// SIMATIC STEP 7 (V5.x) project Gradirn
// CPU: CPU 315-2PN/DP
// station: Hardware
// station: SIMATIC 300(1)
// station: P_ADR_BUS
// station: P_ADR_BUS
// station: Configuration
// program: S7 Program(3)

SYMBOL_TABLE
""		
"grad_motor_1"	DB 1	FB 41
"grad_motor_2"	DB 2	FB 41
"Alarms"	DB 3	DB 3
"values"	DB 4	DB 4
"Data_motors"	DB 5	FB 4
"Motor_grad"	FB 1	FB 1	// Вентилятор градирни
"Motors"	FB 4	FB 4
"CONT_C"	FB 41	FB 41	// Continuous Control
"CONT_S"	FB 42	FB 42	// Step Control
"TCONT_CP"	FB 58	FB 58	// temperature PID controller with pulse generator and self-tuning
"TCONT_S"	FB 59	FB 59	// temperature PID step controller
"Level_grad"	FC 1	FC 1
"read/write values"	FC 2	FC 2
"Fault_motor"	FC 3	FC 3
"Pumps"	FC 4	FC 4
"Alarm"	FC 5	FC 5
"S5TI_TIM"	FC 33	FC 33	// S5 Time to IEC Time
"TIM_S5TI"	FC 40	FC 40	// IEC Time to S5 Time
"Read Analog Value 464-1"	FC 104	FC 104	// Read Analog Value 464-1
"Read Analog Value 464-2"	FC 105	FC 105	// Read Analog Value 464-2
"mode_man_V1"	M 0.0	BOOL
"valve_out"	M 2.0	BOOL
"valve_opened"	M 2.1	BOOL
"valve_closed"	M 2.2	BOOL
"always_on"	M 6.0	BOOL	// всегда 1
"V1_btn_pusk"	M 100.0	BOOL
"V1_btn_stop"	M 100.1	BOOL
"V1_inverter_ok"	M 100.2	BOOL
"V1_mode_remote"	M 100.3	BOOL
"V1_start"	M 100.4	BOOL
"V1_error"	M 100.5	BOOL
"V1_loc_p"	M 100.6	BOOL
"V1_loc_st"	M 100.7	BOOL
"V2_btn_pusk"	M 101.0	BOOL
"V2_btn_stop"	M 101.1	BOOL
"V2_inverter_ok"	M 101.2	BOOL
"V2_mode_remote"	M 101.3	BOOL
"V2_start"	M 101.4	BOOL
"V2_error"	M 101.5	BOOL
"V2_loc_p"	M 101.6	BOOL
"V2_loc_st"	M 101.7	BOOL
"on_H1"	M 102.0	BOOL
"on_H2"	M 102.1	BOOL
"psal_H1"	M 102.2	BOOL
"psal_H2"	M 102.3	BOOL
"tsah_H1"	M 102.4	BOOL
"tsah_H2"	M 102.5	BOOL
"H1_PU"	M 102.6	BOOL
"H1_ST"	M 102.7	BOOL
"H1_MD"	M 103.0	BOOL
"H2_PU"	M 103.1	BOOL
"H2_ST"	M 103.2	BOOL
"H2_MD"	M 103.3	BOOL
"rez_H1"	M 103.4	BOOL
"rez_H2"	M 103.5	BOOL
"btn_H1_PU"	M 103.6	BOOL
"btn_H1_ST"	M 103.7	BOOL
"btn_H2_PU"	M 104.0	BOOL
"btn_H2_ST"	M 104.1	BOOL
"V1_running"	M 110.0	BOOL
"V2_running"	M 111.1	BOOL
"V1_Gain"	MD 2	REAL
"V1_I"	MD 6	TIME
"V1_SP"	MD 10	REAL
"V1_out_freq"	MD 14	REAL
"Temp_grad"	MD 18	REAL
"V1_MAN_SP"	MD 22	REAL
"V_cycle"	MD 26	TIME
"main"	OB 1	OB 1
"pid"	OB 35	OB 35
"TON"	SFB 4	SFB 4	// Generate an On Delay
"Analog values insert"	UDT 1	UDT 1
END_SYMBOL_TABLE

FUNCTION_BLOCK "Motor_grad"	// FB 1
VERSION : 0.1
VAR_INPUT
  btn_pusk : BOOL ;
  btn_stop : BOOL ;
  mode_remote : BOOL ;
  inverter_ok : BOOL ;
  motor_error : BOOL ;
  loc_pusk : BOOL ;
  loc_stop : BOOL ;
  tim_1 : TIMER ;
  tim_2 : TIMER ;
END_VAR
VAR_OUTPUT
  motor_start : BOOL ;
END_VAR
BEGIN
NETWORK
TITLE = start
      A     #inverter_ok;
      A     #mode_remote;
      A     #btn_pusk;
      O(;
      AN    #mode_remote;
      A     #inverter_ok;
      A     #loc_pusk;
      L     S5T#400MS;
      T     LD 0;
      TAK;
      T     LD 4;
      L     #tim_1;
      T     LW 8;
      L     LD 4;
      L     LD 0;
      SD    T [LW 8];
      T     LD 0;
      TAK;
      T     LD 4;
      L     #tim_1;
      T     LW 8;
      L     LD 4;
      L     LD 0;
      A     T [LW 8];
      );
      S     #motor_start;
NETWORK
TITLE = stop
      ON    #inverter_ok;
      O     #motor_error;
      O(;
      A     #mode_remote;
      A     #btn_stop;
      );
      O(;
      L     S5T#400MS;
      AN    #mode_remote;
      A     #loc_stop;
      T     LD 0;
      TAK;
      T     LD 4;
      L     #tim_2;
      T     LW 8;
      L     LD 4;
      L     LD 0;
      SD    T [LW 8];
      T     LD 0;
      TAK;
      T     LD 4;
      L     #tim_2;
      T     LW 8;
      L     LD 4;
      L     LD 0;
      A     T [LW 8];
      );
      R     #motor_start;
END_FUNCTION_BLOCK

FUNCTION_BLOCK "Motors"	// FB 4
VERSION : 0.1
VAR
  mifb_1 : FB 1;
  mifb_2 : FB 1;
END_VAR
BEGIN
NETWORK
TITLE =
      CALL  #mifb_1 (
           btn_pusk                 := "V1_btn_pusk",
           btn_stop                 := "V1_btn_stop",
           mode_remote              := "V1_mode_remote",
           inverter_ok              := "V1_inverter_ok",
           motor_error              := "V1_error",
           loc_pusk                 := "V1_loc_p",
           loc_stop                 := "V1_loc_st",
           tim_1                    := T 1,
           tim_2                    := T 2,
           motor_start              := "V1_start");
NETWORK
TITLE =
      CALL  #mifb_2 (
           btn_pusk                 := "V2_btn_pusk",
           btn_stop                 := "V2_btn_stop",
           mode_remote              := "V2_mode_remote",
           inverter_ok              := "V2_inverter_ok",
           motor_error              := "V2_error",
           loc_pusk                 := "V2_loc_p",
           loc_stop                 := "V2_loc_st",
           tim_1                    := T 3,
           tim_2                    := T 4,
           motor_start              := "V2_start");
END_FUNCTION_BLOCK

// FB 41: know-how protected block, not included

FUNCTION "Level_grad" : VOID	// FC 1
TITLE = Fulling level grad
VERSION : 0.1
BEGIN
NETWORK
TITLE =
      L     "values".level_grad;
      L     "values".level_sp;
      <R;
      JC    open;
      R     "valve_out";
      JU    end;
open: S     "valve_out";
end:  NOP   0;
END_FUNCTION

FUNCTION "read/write values" : VOID	// FC 2
VERSION : 0.1
BEGIN
NETWORK
TITLE =
      A     "values".zero;
      =     L 0.0;
      BLD   103;
      CALL  "Read Analog Value 464-2" (
           $1                       := P#P 256.0,
           $2                       := "values".hi_temp_grad,
           $3                       := "values".low_temp_grad,
           $4                       := L 0.0,
           $5                       := "values".error_temp_grad,
           $6                       := "values".temp_grad);
      NOP   0;
NETWORK
TITLE =
      A     "values".zero;
      =     L 0.0;
      BLD   103;
      CALL  "Read Analog Value 464-2" (
           $1                       := P#P 272.0,
           $2                       := "values".level_hi,
           $3                       := "values".level_low,
           $4                       := L 0.0,
           $5                       := "values".error_level,
           $6                       := "values".level_grad);
      NOP   0;
NETWORK
TITLE = read vibrations motors
      A     "values".zero;
      =     L 0.0;
      BLD   103;
      CALL  "Read Analog Value 464-2" (
           $1                       := P#P 274.0,
           $2                       := "values".vibr_1_hi,
           $3                       := "values".vibr_1_low,
           $4                       := L 0.0,
           $5                       := "values".vibr_1_er,
           $6                       := "values".vibr_1);
      NOP   0;
NETWORK
TITLE =
      A     "values".zero;
      =     L 0.0;
      BLD   103;
      CALL  "Read Analog Value 464-2" (
           $1                       := P#P 276.0,
           $2                       := "values".vibr_1_hi,
           $3                       := "values".vibr_1_low,
           $4                       := L 0.0,
           $5                       := "values".vibr_2_er,
           $6                       := "values".vibr_2);
      NOP   0;
NETWORK
TITLE = Current V1
      CALL  "Read Analog Value 464-2" (
           $1                       := P#P 278.0,
           $2                       := "values".curr_1_hi,
           $3                       := "values".curr_1_low,
           $4                       := "values".zero,
           $5                       := "values".curr_1_er,
           $6                       := "values".curr_1);
NETWORK
TITLE = Current V2
      CALL  "Read Analog Value 464-2" (
           $1                       := P#P 280.0,
           $2                       := "values".curr_1_hi,
           $3                       := "values".curr_1_low,
           $4                       := "values".zero,
           $5                       := "values".curr_2_er,
           $6                       := "values".curr_2);
NETWORK
TITLE = discret inputs/outputs V1,V2
      A     I 8.0;
      =     "V1_loc_p";
      A     I 8.1;
      =     "V1_loc_st";
      A     I 8.2;
      =     "V1_inverter_ok";
      A     "V1_start";
      =     Q 11.0;
      A     I 8.3;
      =     "V1_mode_remote";
      A     I 8.4;
      =     "V1_running";
      A     I 9.0;
      =     "V2_loc_p";
      A     I 9.1;
      =     "V2_loc_st";
      A     I 9.2;
      =     "V2_inverter_ok";
      A     "V2_start";
      =     Q 11.1;
      A     I 9.3;
      =     "V2_mode_remote";
      A     I 9.4;
      =     "V2_running";
NETWORK
TITLE = Pump signals
      A     I 10.0;
      =     "on_H1";
      A     I 10.1;
      =     "on_H2";
      A     I 10.2;
      =     "psal_H1";
      A     I 10.3;
      =     "psal_H2";
      A     I 10.4;
      =     "tsah_H1";
      A     I 10.5;
      =     "tsah_H2";
      A     "H1_PU";
      =     Q 11.2;
      A     "H1_ST";
      =     Q 11.3;
      A     "H1_MD";
      =     Q 11.4;
      A     "H2_PU";
      =     Q 11.5;
      A     "H2_ST";
      =     Q 11.6;
      A     "H2_MD";
      =     Q 11.7;
NETWORK
TITLE =
      CALL  "Read Analog Value 464-2" (
           $1                       := P#P 282.0,
           $2                       := "values".curr_1_hi,
           $3                       := "values".curr_1_low,
           $4                       := "values".zero,
           $5                       := "values".curr_H1_er,
           $6                       := "values".curr_H1);
      CALL  "Read Analog Value 464-2" (
           $1                       := P#P 284.0,
           $2                       := "values".curr_1_hi,
           $3                       := "values".curr_1_low,
           $4                       := "values".zero,
           $5                       := "values".curr_H2_er,
           $6                       := "values".curr_2);
END_FUNCTION

FUNCTION "Fault_motor" : VOID	// FC 3
VERSION : 0.1
BEGIN
NETWORK
TITLE = fault motor 1 of vibration
      L     "values".vibr_1;
      L     1.200000e+01;
      >R;
      =     "V1_error";
NETWORK
TITLE =
      L     "values".vibr_2;
      L     1.200000e+01;
      >R;
      =     "V2_error";
END_FUNCTION

FUNCTION "Pumps" : VOID	// FC 4
VERSION : 0.1
VAR_TEMP
  fl_1 : BOOL ;
  fl_2 : BOOL ;
  tr_1 : BOOL ;
END_VAR
BEGIN
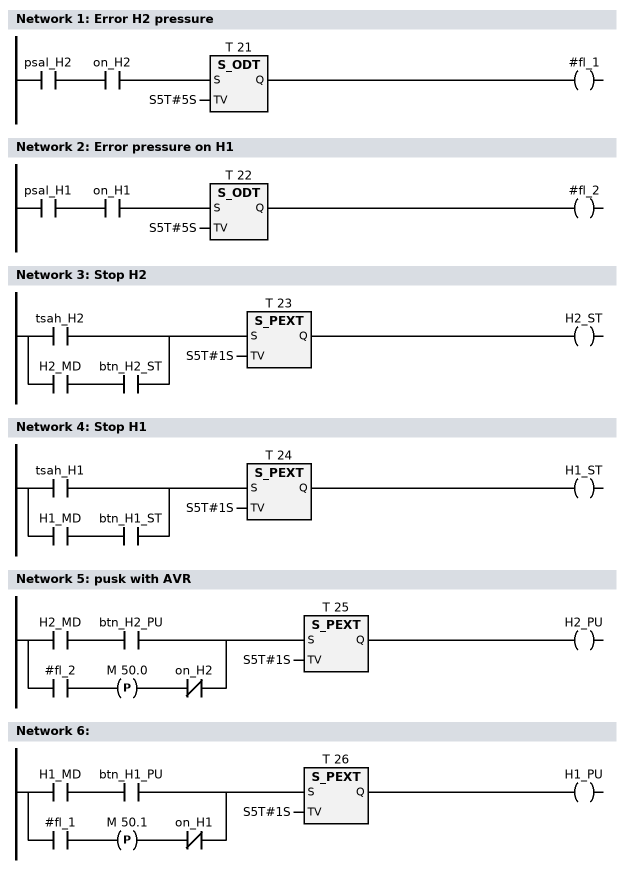
NETWORK
TITLE = Error H2 pressure
      A     "psal_H2";
      A     "on_H2";
      L     S5T#5S;
      SD    T 21;
      NOP   0;
      NOP   0;
      NOP   0;
      A     T 21;
      =     #fl_1;
NETWORK
TITLE = Error pressure on H1
      A     "psal_H1";
      A     "on_H1";
      L     S5T#5S;
      SD    T 22;
      NOP   0;
      NOP   0;
      NOP   0;
      A     T 22;
      =     #fl_2;
NETWORK
TITLE = Stop H2
      A(;
      O     "tsah_H2";
      O;
      A     "H2_MD";
      A     "btn_H2_ST";
      );
      L     S5T#1S;
      SE    T 23;
      NOP   0;
      NOP   0;
      NOP   0;
      A     T 23;
      =     "H2_ST";
NETWORK
TITLE = Stop H1
      A(;
      O     "tsah_H1";
      O;
      A     "H1_MD";
      A     "btn_H1_ST";
      );
      L     S5T#1S;
      SE    T 24;
      NOP   0;
      NOP   0;
      NOP   0;
      A     T 24;
      =     "H1_ST";
NETWORK
TITLE = pusk with AVR
      A(;
      A     "H2_MD";
      A     "btn_H2_PU";
      O(;
      A     #fl_2;
      FP    M 50.0;
      AN    "on_H2";
      );
      );
      L     S5T#1S;
      SE    T 25;
      NOP   0;
      NOP   0;
      NOP   0;
      A     T 25;
      =     "H2_PU";
NETWORK
TITLE =
      A(;
      A     "H1_MD";
      A     "btn_H1_PU";
      O(;
      A     #fl_1;
      FP    M 50.1;
      AN    "on_H1";
      );
      );
      L     S5T#1S;
      SE    T 26;
      NOP   0;
      NOP   0;
      NOP   0;
      A     T 26;
      =     "H1_PU";
END_FUNCTION

FUNCTION "Alarm" : VOID	// FC 5
VERSION : 0.1
BEGIN
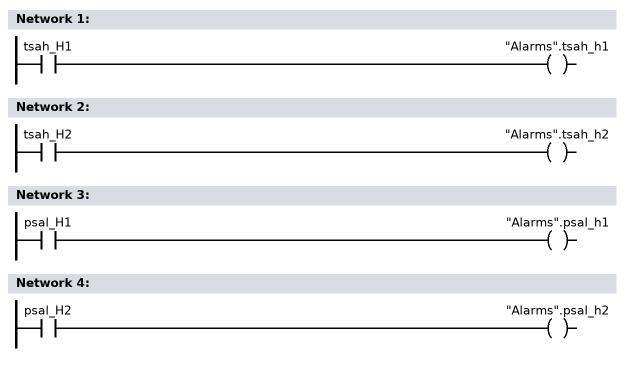
NETWORK
TITLE =
      A     "tsah_H1";
      =     "Alarms".tsah_h1;
NETWORK
TITLE =
      A     "tsah_H2";
      =     "Alarms".tsah_h2;
NETWORK
TITLE =
      A     "psal_H1";
      =     "Alarms".psal_h1;
NETWORK
TITLE =
      A     "psal_H2";
      =     "Alarms".psal_h2;
END_FUNCTION

FUNCTION FC 6 : VOID
VERSION : 0.1
BEGIN
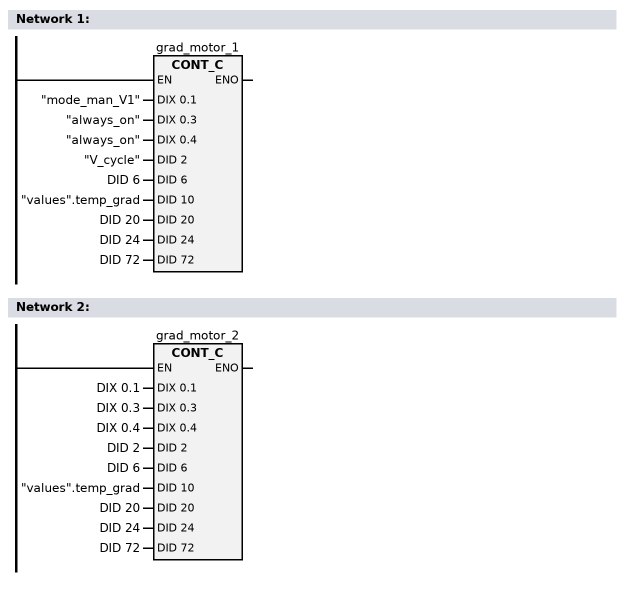
NETWORK
TITLE =
      CALL  "CONT_C" , "grad_motor_1" (
           DIX 0.1                  := "mode_man_V1",
           DIX 0.3                  := "always_on",
           DIX 0.4                  := "always_on",
           DID 2                    := "V_cycle",
           DID 6                    := DID 6,
           DID 10                   := "values".temp_grad,
           DID 20                   := DID 20,
           DID 24                   := DID 24,
           DID 72                   := DID 72);
NETWORK
TITLE =
      CALL  "CONT_C" , "grad_motor_2" (
           DIX 0.1                  := DIX 0.1,
           DIX 0.3                  := DIX 0.3,
           DIX 0.4                  := DIX 0.4,
           DID 2                    := DID 2,
           DID 6                    := DID 6,
           DID 10                   := "values".temp_grad,
           DID 20                   := DID 20,
           DID 24                   := DID 24,
           DID 72                   := DID 72);
END_FUNCTION

// FC 33: know-how protected block, not included

// FC 40: know-how protected block, not included

// FC 105: know-how protected block, not included

DATA_BLOCK "grad_motor_1"	// DB 1
AUTHOR : SIMATIC
FAMILY : ICONT
VERSION : 0.1
"CONT_C"
BEGIN
END_DATA_BLOCK

DATA_BLOCK "grad_motor_2"	// DB 2
AUTHOR : SIMATIC
FAMILY : ICONT
VERSION : 0.1
"CONT_C"
BEGIN
END_DATA_BLOCK

DATA_BLOCK "Alarms"	// DB 3
VERSION : 0.1
  STRUCT
   tsah_h1 : BOOL ;
   tsah_h2 : BOOL ;
   psal_h1 : BOOL ;
   psal_h2 : BOOL ;
  END_STRUCT ;	
BEGIN
END_DATA_BLOCK

DATA_BLOCK "values"	// DB 4
VERSION : 0.1
  STRUCT
   hi_temp_grad : REAL  := 1.000000e+002;
   low_temp_grad : REAL ;
   zero : BOOL ;
   temp_grad : REAL ;
   error_temp_grad : WORD ;
   level_hi : REAL  := 1.000000e+002;
   level_low : REAL ;
   level_grad : REAL ;
   error_level : WORD ;
   level_sp : REAL ;
   vibr_1_low : REAL ;
   vibr_1_hi : REAL  := 4.000000e+001;
   vibr_1_er : WORD ;
   vibr_1 : REAL ;
   vibr_2_er : WORD ;
   vibr_2 : REAL ;
   curr_1_low : REAL ;
   curr_1_hi : REAL  := 5.000000e+001;
   curr_1_er : WORD ;
   curr_1 : REAL ;
   curr_2_er : WORD ;
   curr_2 : REAL ;
   curr_H1 : REAL ;
   curr_H2 : REAL ;
   curr_H1_er : WORD ;
   curr_H2_er : WORD ;
  END_STRUCT ;	
BEGIN
   hi_temp_grad := 1.000000e+02;
   level_hi := 1.000000e+02;
   level_sp := 9.000000e+01;
   vibr_1_hi := 4.000000e+01;
   curr_1_hi := 5.000000e+01;
END_DATA_BLOCK

DATA_BLOCK "Data_motors"	// DB 5
VERSION : 0.0
"Motors"
BEGIN
END_DATA_BLOCK

DATA_BLOCK DB 12
AUTHOR : SIMATIC
FAMILY : IEC_TC
VERSION : 0.0
"TON"
BEGIN
END_DATA_BLOCK

ORGANIZATION_BLOCK "main"	// OB 1
TITLE = "Main Program Sweep (Cycle)"
VERSION : 0.1
VAR_TEMP
  OB1_EV_CLASS : BYTE ;	//Bits 0-3 = 1 (Coming event), Bits 4-7 = 1 (Event class 1)
  OB1_SCAN_1 : BYTE ;	//1 (Cold restart scan 1 of OB 1), 3 (Scan 2-n of OB 1)
  OB1_PRIORITY : BYTE ;	//Priority of OB Execution
  OB1_OB_NUMBR : BYTE ;	//1 (Organization block 1, OB1)
  OB1_RESERVED_1 : BYTE ;	//Reserved for system
  OB1_RESERVED_2 : BYTE ;	//Reserved for system
  OB1_PREV_CYCLE : INT ;	//Cycle time of previous OB1 scan (milliseconds)
  OB1_MIN_CYCLE : INT ;	//Minimum cycle time of OB1 (milliseconds)
  OB1_MAX_CYCLE : INT ;	//Maximum cycle time of OB1 (milliseconds)
  OB1_DATE_TIME : DATE_AND_TIME ;	//Date and time OB1 started
END_VAR
BEGIN
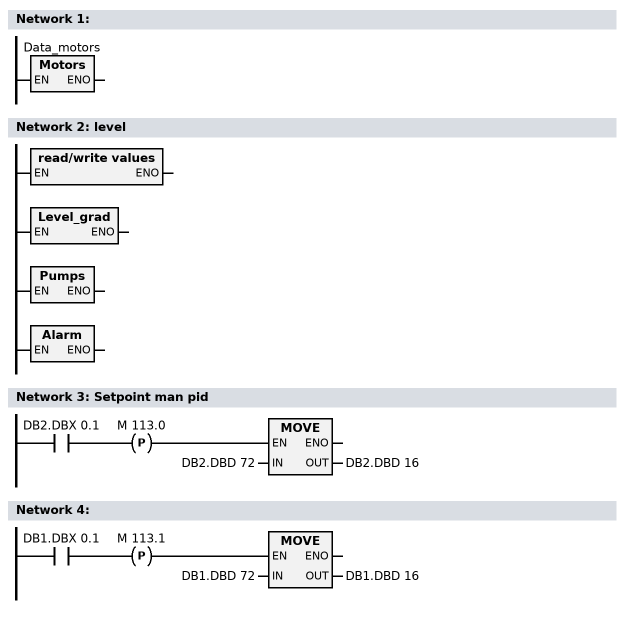
NETWORK
TITLE =
      CALL  "Motors" , "Data_motors";
NETWORK
TITLE = level
      CALL  "read/write values";
      CALL  "Level_grad";
      CALL  "Pumps";
      CALL  "Alarm";
NETWORK
TITLE = Setpoint man pid
      A     DB2.DBX 0.1;
      FP    M 113.0;
      JNB   _001;
      L     DB2.DBD 72;
      T     DB2.DBD 16;
_001: NOP   0;
NETWORK
TITLE =
      A     DB1.DBX 0.1;
      FP    M 113.1;
      JNB   _002;
      L     DB1.DBD 72;
      T     DB1.DBD 16;
_002: NOP   0;
END_ORGANIZATION_BLOCK

ORGANIZATION_BLOCK "pid"	// OB 35
TITLE = "Cyclic Interrupt"
VERSION : 0.1
VAR_TEMP
  OB35_EV_CLASS : BYTE ;	//Bits 0-3 = 1 (Coming event), Bits 4-7 = 1 (Event class 1)
  OB35_STRT_INF : BYTE ;	//16#36 (OB 35 has started)
  OB35_PRIORITY : BYTE ;	//Priority of OB Execution
  OB35_OB_NUMBR : BYTE ;	//35 (Organization block 35, OB35)
  OB35_RESERVED_1 : BYTE ;	//Reserved for system
  OB35_RESERVED_2 : BYTE ;	//Reserved for system
  OB35_PHASE_OFFSET : WORD ;	//Phase offset (msec)
  OB35_RESERVED_3 : INT ;	//Reserved for system
  OB35_EXC_FREQ : INT ;	//Frequency of execution (msec)
  OB35_DATE_TIME : DATE_AND_TIME ;	//Date and time OB35 started
END_VAR
BEGIN
NETWORK
TITLE =
      CALL  "CONT_C" , "grad_motor_1" (
           DIX 0.1                  := DIX 0.1,
           DIX 0.3                  := DIX 0.3,
           DIX 0.4                  := DIX 0.4,
           DID 2                    := DID 2,
           DID 6                    := DID 6,
           DID 10                   := "values".temp_grad,
           DID 20                   := DID 20,
           DID 24                   := DID 24,
           DID 72                   := DID 72);
NETWORK
TITLE =
      CALL  "CONT_C" , "grad_motor_2" (
           DIX 0.1                  := DIX 0.1,
           DIX 0.3                  := DIX 0.3,
           DIX 0.4                  := DIX 0.4,
           DID 2                    := DID 2,
           DID 6                    := DID 6,
           DID 10                   := "values".temp_grad,
           DID 20                   := DID 20,
           DID 24                   := DID 24,
           DID 72                   := DID 72);
END_ORGANIZATION_BLOCK
